(* IEC 61131-3 sources: repolevel_ST_code_completion/output/full_case_fixed/repoeval_electronic_gear_motion/readful_result, 3 files *)

(* ---- FB_DualAxisPower.st ---- *)
FUNCTION_BLOCK FB_DualAxisPower
VAR_INPUT
	Axis1			:	AXIS_REF;		//轴1引用
	Axis2			:	AXIS_REF;		//轴2引用
	bEnable			:	BOOL := TRUE;	//使能信号
END_VAR
VAR_OUTPUT
	bAxis1Ready		:	BOOL;			//轴1准备就绪
	bAxis2Ready		:	BOOL;			//轴2准备就绪
	bBothReady		:	BOOL;			//两轴都准备就绪
	bError			:	BOOL;			//错误标志
END_VAR
VAR
	fbPower1		:	MC_Power;		//轴1电源控制
	fbPower2		:	MC_Power;		//轴2电源控制
	bAxis1Error		:	BOOL;			//轴1错误标志
	bAxis2Error		:	BOOL;			//轴2错误标志
END_VAR

fbPower1(
 Axis := Axis1,
 Enable := bEnable
);

fbPower2(
 Axis := Axis2,
 Enable := bEnable
);

// Assuming correct logic for readiness is "Status = TRUE"
bAxis1Ready := fbPower1.Status = MC_POWER_READY;
bAxis2Ready := fbPower2.Status = MC_POWER_READY;

bAxis1Error := fbPower1.Error;
bAxis2Error := fbPower2.Error;

bError := bAxis1Error OR bAxis2Error;

bBothReady := bAxis1Ready AND bAxis2Ready;
END_FUNCTION_BLOCK

(* ---- FB_GearCoupling.st ---- *)
FUNCTION_BLOCK FB_GearCoupling
VAR_INPUT
	Master				:	AXIS_REF;		//主轴引用
	Slave				:	AXIS_REF;		//从轴引用
	bCouple				:	BOOL;			//TRUE=耦合，FALSE=解耦
	nRatioNumerator		:	INT := 1;		//传动比分子
	nRatioDenominator	:	INT := 1;		//传动比分母
	rAcceleration		:	REAL := 10000.0;//加速度
	rDeceleration		:	REAL := 10000.0;//减速度
END_VAR
VAR_OUTPUT
	bInGear				:	BOOL;			//耦合状态
	bCouplingDone		:	BOOL;			//耦合完成
	bDecouplingDone		:	BOOL;			//解耦完成
	bError				:	BOOL;			//错误标志
	nErrorID			:	DWORD;			//错误代码
END_VAR
VAR
	fbGearIn			:	MC_GearIn;		//齿轮耦合功能块
	fbGearOut			:	MC_GearOut;		//齿轮解耦功能块
	bLastCouple			:	BOOL;			//上次耦合状态
	bCoupleRising		:	BOOL;			//耦合上升沿
	bCoupleFalling		:	BOOL;			//耦合下降沿
END_VAR

// 检测耦合信号的边沿
bCoupleRising := bCouple AND NOT bLastCouple;
bCoupleFalling := NOT bCouple AND bLastCouple;
bLastCouple := bCouple;

// 耦合逻辑
IF bCoupleRising THEN
 fbGearIn.Master := Master;
 fbGearIn.Slave := Slave;
 fbGearIn.RatioNumerator := nRatioNumerator;
 fbGearIn.RatioDenominator := nRatioDenominator;
 fbGearIn.Acceleration := rAcceleration;
 fbGearIn.Execute := TRUE; // Start the gear-in operation
END_IF;

// 检查耦合完成或错误状态
IF fbGearIn.Execute THEN
 IF fbGearIn.Done THEN
  bInGear := TRUE;
  bCouplingDone := TRUE;
  fbGearIn.Execute := FALSE; // Reset Execute to stop operation
 ELSIF fbGearIn.Error THEN
  bError := TRUE;
  nErrorID := fbGearIn.ErrorID;
  fbGearIn.Execute := FALSE; // Reset Execute on error
 END_IF;
END_IF;

// 解耦逻辑
IF bCoupleFalling THEN
 fbGearOut.Slave := Slave;
 fbGearOut.Execute := TRUE; // Start the gear-out operation
END_IF;

// 检查解耦完成或错误状态
IF fbGearOut.Execute THEN
 IF fbGearOut.Done THEN
  bInGear := FALSE;
  bDecouplingDone := TRUE;
  fbGearOut.Execute := FALSE; // Reset Execute to stop operation
 ELSIF fbGearOut.Error THEN
  bError := TRUE;
  nErrorID := fbGearOut.ErrorID;
  fbGearOut.Execute := FALSE; // Reset Execute on error
 END_IF;
END_IF;
END_FUNCTION_BLOCK

(* ---- FB_GearMotionControl.st ---- *)
FUNCTION_BLOCK FB_GearMotionControl
VAR_INPUT
	MasterAxis			:	AXIS_REF;		//主轴引用
	SlaveAxis			:	AXIS_REF;		//从轴引用
	bStart				:	BOOL;			//启动信号
	bStop				:	BOOL;			//停止信号
	nRatioNumerator		:	INT := 1;		//传动比分子
	nRatioDenominator	:	INT := 1;		//传动比分母
	nDirection			:	INT := 1;		//运动方向（1=正向，-1=反向）
	rVelocity			:	REAL := 360.0;	//主轴速度
	rAcceleration		:	REAL := 10000.0;//加速度
	rDeceleration		:	REAL := 10000.0;//减速度
END_VAR
VAR_OUTPUT
	bRunning			:	BOOL;			//运行中
	bReady				:	BOOL;			//准备就绪（可以启动）
	bError				:	BOOL;			//错误标志
	nCurrentState		:	BYTE;			//当前状态
END_VAR
VAR
	fbPowerMgr			:	FB_DualAxisPower;	//双轴电源管理
	fbGearCtrl			:	FB_GearCoupling;	//齿轮耦合控制
	fbMoveVel			:	MC_MoveVelocity;	//速度运动
	fbHaltMaster		:	MC_Halt;			//主轴停止
	fbHaltSlave			:	MC_Halt;			//从轴停止
	fbStartRtrig		:	R_TRIG;				//启动上升沿
	fbStopRtrig			:	R_TRIG;				//停止上升沿
	nState				:	BYTE;				//内部状态机
END_VAR

fbPowerMgr(
	Axis1 := MasterAxis,
	Axis2 := SlaveAxis,
	bEnable := TRUE
);

fbStartRtrig(CLK := bStart);
fbStopRtrig(CLK := bStop);

CASE nState OF
	0: // 等待轴准备就绪
		IF fbPowerMgr.bReady THEN
			bReady := TRUE;
			nState := 1;
		END_IF;

	1: // 启动运动
		IF fbStartRtrig.Q THEN
fbMoveVel(
Axis := MasterAxis,
Velocity := rVelocity,
Acceleration := rAcceleration,
Deceleration := rDeceleration,
Direction := BOOL_TO_DINT(nDirection),
Execute := TRUE
); // Ensure the `Direction` uses the correct data type conversion
			IF fbMoveVel.Done THEN
fbGearCtrl(
Master := MasterAxis,
Slave := SlaveAxis,
RatioNumerator := DINT_TO_REAL(nRatioNumerator),
RatioDenominator := DINT_TO_REAL(nRatioDenominator),
Execute := TRUE
); // Ensure proper data types for Ratios
				IF fbGearCtrl.Done THEN
					bRunning := TRUE;
					nState := 2;
				END_IF;
			END_IF;
		END_IF;

	2: // 运行中
		IF fbStopRtrig.Q THEN
fbHaltMaster(
Axis := MasterAxis,
Execute := TRUE
); // Clean function call without inline comments

fbHaltSlave(
Axis := SlaveAxis,
Execute := TRUE
); // Clean function call without inline comments
			IF fbHaltMaster.Done AND fbHaltSlave.Done THEN
				bRunning := FALSE;
				nState := 0;
			END_IF;
		END_IF;

	ELSE
		bError := TRUE;
END_CASE;

nCurrentState := nState;
END_FUNCTION_BLOCK
